// TIA Portal project "Vyrobne_kleman_Omdrejka_1.1" (V15.1)

(* hardware
DEVICE "S7-1200 station_1"  S7-1200 Station
   slot 0: "Rack_0"  S7-1200 Rack  Rack  V1.0
   slot 1: "PLC_1"  CPU 1215C DC/DC/DC  6ES7 215-1AG40-0XB0  V4.2
*)

// ===== PLC "PLC_1"  CPU 1215C DC/DC/DC =====

VAR_GLOBAL   // PLC tag table "dig_IN"
   "KS1_VZ" AT %I0.0 : Bool;   // posuvnik 1 zadne TL
   "KS1_VP" AT %I0.1 : Bool;
   "KS2_VP" AT %I0.2 : Bool;
   "KS2_VZ" AT %I0.3 : Bool;
   "OS1" AT %I0.4 : Bool;
   "OS2" AT %I0.5 : Bool;
   "T_LOAD" AT %I0.6 : Bool;
   "OS3" AT %I0.7 : Bool;
   "OS4" AT %I1.0 : Bool;
END_VAR

VAR_GLOBAL   // PLC tag table "dig_OUT"
   "P1_VZ" AT %Q0.0 : Bool;
   "P1_VP" AT %Q0.1 : Bool;
   "P2_VP" AT %Q0.2 : Bool;
   "P2_VZ" AT %Q0.3 : Bool;
   "D1" AT %Q0.4 : Bool;
   "D2" AT %Q0.5 : Bool;
   "S1" AT %Q0.6 : Bool;
   "D3" AT %Q0.7 : Bool;
   "S2" AT %Q1.0 : Bool;
   "D4" AT %Q1.1 : Bool;
END_VAR

VAR_GLOBAL   // PLC tag table "pomocne_premenne"
   "Pos_START" AT %M0.0 : Bool;
   "Pos1" AT %M0.1 : Bool;
   "Pos2" AT %M0.2 : Bool;
   "Pos3" AT %M0.3 : Bool;
   "Pos4" AT %M0.4 : Bool;
   "PosP" AT %M0.7 : Bool;
   "S1_pracuje" AT %M1.0 : Bool;
   "S1_dopracoval" AT %M1.1 : Bool;
   "S2_pracuje" AT %M1.3 : Bool;
   "S2_dopracoval" AT %M1.4 : Bool;
   "PosStart_id" AT %MW4 : Int;   // ID na zaciatku D1 po potvrdeni nalozenia
   "Pos1_id" AT %MW6 : Int;   // ID na linke 0 = prazdne
   "PosP_id" AT %MW8 : Int;   // ID na linke 0 = prazdne
   "Pos2_id" AT %MW10 : Int;   // ID na linke 0 = prazdne
   "Pos3_id" AT %MW12 : Int;   // ID na linke 0 = prazdne
   "Pos4_id" AT %MW14 : Int;   // ID na linke 0 = prazdne
   "Ptrig_1" AT %M20.0 : Bool;   // T_LOAD
   "Ptrig_2" AT %M20.1 : Bool;   // prerusenie OS1
   "Ptrig_3" AT %M20.2 : Bool;   // prerusenie OS2
   "Ptrig_4" AT %M20.3 : Bool;   // reset_CTU_1
   "ptrig_5" AT %M20.5 : Bool;   // OS3
   "ptrig_6" AT %M20.6 : Bool;   // Reset_CTU_S2
   "ptrig_7" AT %M20.7 : Bool;   // OS4
   "ptrig_8" AT %M21.0 : Bool;   // krok_1
   "ptrig_9" AT %M21.1 : Bool;   // pos_4==2
   "ptrig_10" AT %M21.2 : Bool;   // krok_4
   "ptrig_11" AT %M21.3 : Bool;   // posStart_r
   "ptrig_12" AT %M21.4 : Bool;   // pos1_r
   "ptrig_13" AT %M21.5 : Bool;   // posp_r
   "ptrig_14" AT %M21.6 : Bool;   // pos2_r
   "ptrig_15" AT %M21.7 : Bool;   // pos3_r
   "krok" AT %MW22 : Int;   // cislo kroku triedenia
END_VAR

DATA_BLOCK "DB_premenne"   // DB12
{ S7_Optimized_Access := 'TRUE' }
VERSION : 0.1
   VAR RETAIN
      ID_objekt : Int := 1;
      S1_cyklus : Int := 2;
      S2_cyklus : Int := 2;
   END_VAR
BEGIN
END_DATA_BLOCK

// folder: System blocks/Program resources

DATA_BLOCK "IEC_Timer_0_DB"   // DB1
{ S7_Optimized_Access := 'TRUE' }
AUTHOR : Simatic
FAMILY : IEC
NAME : IEC_TMR
VERSION : 1.0
// stored: InstanceOfName IEC_TIMER
"IEC_TIMER"
BEGIN
END_DATA_BLOCK

DATA_BLOCK "casovac_D1_na_PosP"   // DB2
{ S7_Optimized_Access := 'TRUE' }
AUTHOR : Simatic
FAMILY : IEC
NAME : IEC_TMR
VERSION : 1.0
// stored: InstanceOfName IEC_TIMER
"IEC_TIMER"
BEGIN
END_DATA_BLOCK

DATA_BLOCK "IEC_Timer_0_DB_1"   // DB3
{ S7_Optimized_Access := 'TRUE' }
AUTHOR : Simatic
FAMILY : IEC
NAME : IEC_TMR
VERSION : 1.0
// stored: InstanceOfName IEC_TIMER
"IEC_TIMER"
BEGIN
END_DATA_BLOCK

DATA_BLOCK "timer_S2_S"   // DB4
{ S7_Optimized_Access := 'TRUE' }
AUTHOR : Simatic
FAMILY : IEC
NAME : IEC_TMR
VERSION : 1.0
// stored: InstanceOfName IEC_TIMER
"IEC_TIMER"
BEGIN
END_DATA_BLOCK

DATA_BLOCK "timer_S2_R"   // DB5
{ S7_Optimized_Access := 'TRUE' }
AUTHOR : Simatic
FAMILY : IEC
NAME : IEC_TMR
VERSION : 1.0
// stored: InstanceOfName IEC_TIMER
"IEC_TIMER"
BEGIN
END_DATA_BLOCK

DATA_BLOCK "Rpocet_cyklov2"   // DB6
{ S7_Optimized_Access := 'TRUE' }
AUTHOR : Simatic
FAMILY : IEC
NAME : CNTR
VERSION : 1.0
// stored: InstanceOfName IEC_COUNTER
"IEC_COUNTER"
BEGIN
END_DATA_BLOCK

DATA_BLOCK "Rpocet_cyklov1"   // DB7
{ S7_Optimized_Access := 'TRUE' }
AUTHOR : Simatic
FAMILY : IEC
NAME : CNTR
VERSION : 1.0
// stored: InstanceOfName IEC_COUNTER
"IEC_COUNTER"
BEGIN
END_DATA_BLOCK

DATA_BLOCK "IEC_Timer_0_DB_2"   // DB8
{ S7_Optimized_Access := 'TRUE' }
AUTHOR : Simatic
FAMILY : IEC
NAME : IEC_TMR
VERSION : 1.0
// stored: InstanceOfName IEC_TIMER
"IEC_TIMER"
BEGIN
END_DATA_BLOCK

DATA_BLOCK "IEC_Timer_0_DB_3"   // DB9
{ S7_Optimized_Access := 'TRUE' }
AUTHOR : Simatic
FAMILY : IEC
NAME : IEC_TMR
VERSION : 1.0
// stored: InstanceOfName IEC_TIMER
"IEC_TIMER"
BEGIN
END_DATA_BLOCK

DATA_BLOCK "IEC_Timer_0_DB_4"   // DB10
{ S7_Optimized_Access := 'TRUE' }
AUTHOR : Simatic
FAMILY : IEC
NAME : IEC_TMR
VERSION : 1.0
// stored: InstanceOfName IEC_TIMER
"IEC_TIMER"
BEGIN
END_DATA_BLOCK

DATA_BLOCK "IEC_Timer_0_DB_5"   // DB11
{ S7_Optimized_Access := 'TRUE' }
AUTHOR : Simatic
FAMILY : IEC
NAME : IEC_TMR
VERSION : 1.0
// stored: InstanceOfName IEC_TIMER
"IEC_TIMER"
BEGIN
END_DATA_BLOCK

// folder: (top level)

ORGANIZATION_BLOCK "Main"   // OB1, LAD, ProgramCycle
TITLE = "Main Program Sweep (Cycle)"
{ S7_Optimized_Access := 'TRUE' }
VERSION : 0.1
   VAR_INPUT
      Initial_Call : Bool;   // Initial call of this OB
      Remanence : Bool;   // =True, if remanent data are available
   END_VAR
   VAR_TEMP   // added for the SCL form of the ladder/FBD networks
      _w1 : Bool;
      _w2 : Bool;
      _w3 : Bool;
      _w4 : Bool;
      _w5 : Bool;
      _w6 : Bool;
      _w7 : Bool;
      _w8 : Bool;
      _w9 : Bool;
   END_VAR
BEGIN

REGION Network 1: D1 nalozenie
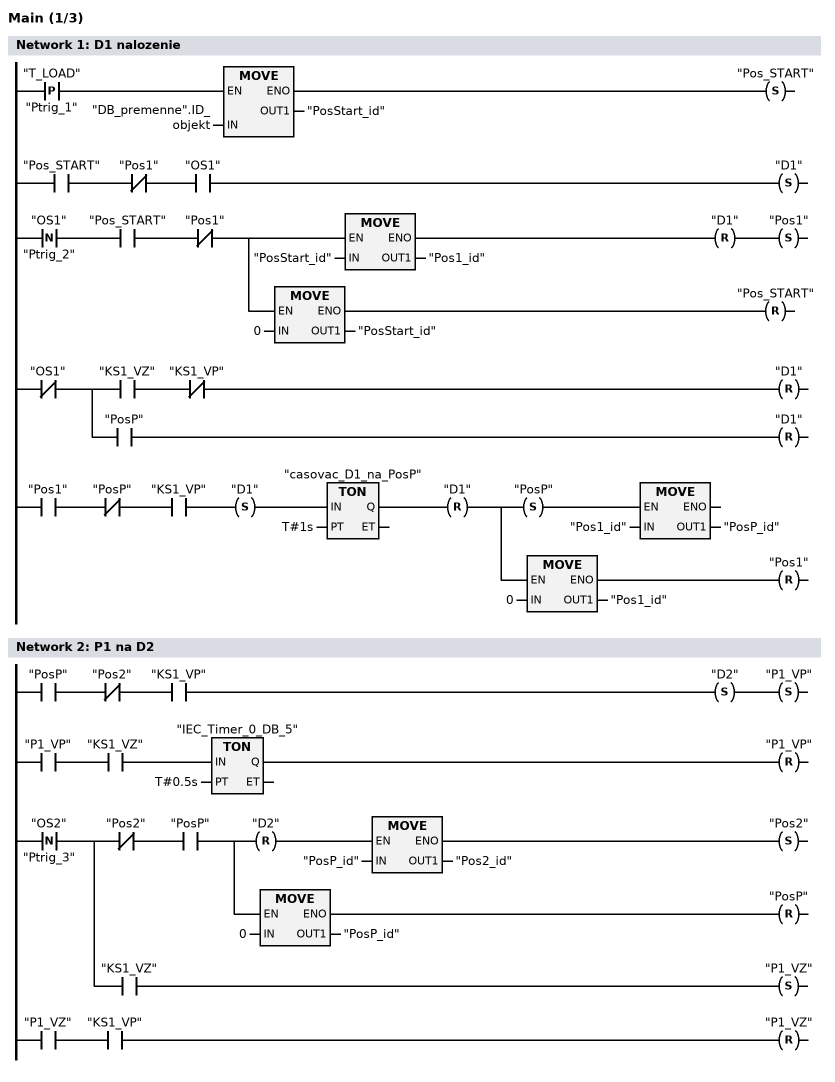
   #_w1 := "T_LOAD" AND NOT "Ptrig_1";   // rising edge of "T_LOAD"
   "Ptrig_1" := "T_LOAD";
   IF #_w1 THEN
       "PosStart_id" := "DB_premenne".ID_objekt;
       "Pos_START" := TRUE;
   END_IF;
   IF "Pos_START" AND NOT "Pos1" AND "OS1" THEN "D1" := TRUE; END_IF;
   #_w2 := NOT "OS1" AND "Ptrig_2";   // falling edge of "OS1"
   "Ptrig_2" := "OS1";
   IF #_w2 AND "Pos_START" AND NOT "Pos1" THEN
       "Pos1_id" := "PosStart_id";
       "D1" := FALSE;
   END_IF;
   #_w3 := #_w2 AND "Pos_START" AND NOT "Pos1";
   IF #_w3 THEN
       "Pos1" := TRUE;
       "PosStart_id" := 0;
       "Pos_START" := FALSE;
   END_IF;
   IF NOT "OS1" AND "KS1_VZ" AND NOT "KS1_VP" THEN "D1" := FALSE; END_IF;
   IF NOT "OS1" AND "PosP" THEN "D1" := FALSE; END_IF;
   #_w4 := "Pos1" AND NOT "PosP" AND "KS1_VP";
   IF #_w4 THEN "D1" := TRUE; END_IF;
   "casovac_D1_na_PosP".TON(IN := #_w4, PT := T#1s);
   IF "casovac_D1_na_PosP".Q THEN
       "D1" := FALSE;
       "PosP" := TRUE;
       "PosP_id" := "Pos1_id";
       "Pos1_id" := 0;
       "Pos1" := FALSE;
   END_IF;
END_REGION

REGION Network 2: P1 na D2
   IF "PosP" AND NOT "Pos2" AND "KS1_VP" THEN
       "D2" := TRUE;
       "P1_VP" := TRUE;
   END_IF;
   "IEC_Timer_0_DB_5".TON(IN := "P1_VP" AND "KS1_VZ", PT := T#0.5s);
   IF "IEC_Timer_0_DB_5".Q THEN "P1_VP" := FALSE; END_IF;
   #_w1 := NOT "OS2" AND "Ptrig_3";   // falling edge of "OS2"
   "Ptrig_3" := "OS2";
   IF #_w1 AND NOT "Pos2" AND "PosP" THEN
       "D2" := FALSE;
       "Pos2_id" := "PosP_id";
   END_IF;
   #_w2 := #_w1 AND NOT "Pos2" AND "PosP";
   IF #_w2 THEN
       "Pos2" := TRUE;
       "PosP_id" := 0;
       "PosP" := FALSE;
   END_IF;
   IF #_w1 AND "KS1_VZ" THEN "P1_VZ" := TRUE; END_IF;
   IF "P1_VZ" AND "KS1_VP" THEN "P1_VZ" := FALSE; END_IF;
END_REGION

REGION Network 3: S1
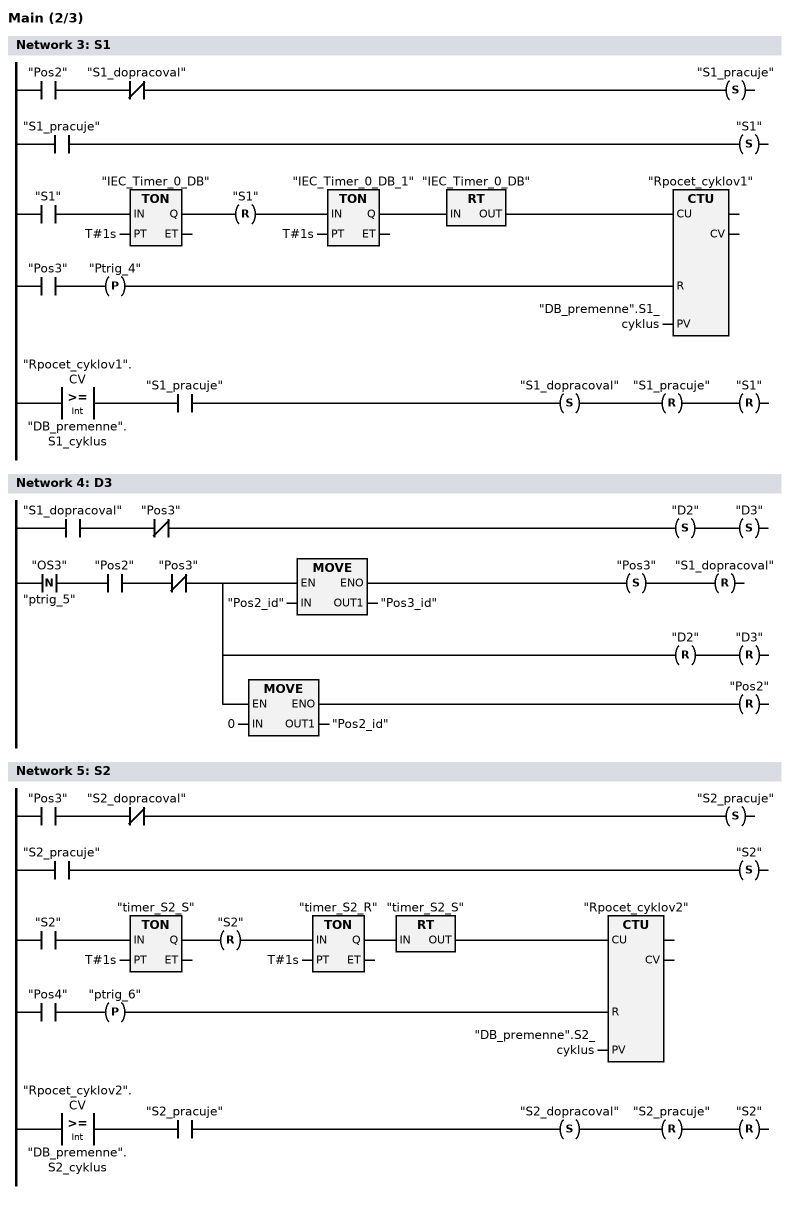
   IF "Pos2" AND NOT "S1_dopracoval" THEN "S1_pracuje" := TRUE; END_IF;
   IF "S1_pracuje" THEN "S1" := TRUE; END_IF;
   "IEC_Timer_0_DB".TON(IN := "S1", PT := T#1s);
   IF "IEC_Timer_0_DB".Q THEN "S1" := FALSE; END_IF;
   "IEC_Timer_0_DB_1".TON(IN := "IEC_Timer_0_DB".Q, PT := T#1s);
   IF "IEC_Timer_0_DB_1".Q THEN RESET_TIMER("IEC_Timer_0_DB"); END_IF;
   #_w1 := "Pos3" AND NOT "Ptrig_4";   // rising edge
   "Ptrig_4" := "Pos3";
   "Rpocet_cyklov1".CTU(CU := "IEC_Timer_0_DB_1".Q, R := #_w1, PV := "DB_premenne".S1_cyklus);
   IF ("Rpocet_cyklov1".CV >= "DB_premenne".S1_cyklus) AND "S1_pracuje" THEN "S1_dopracoval" := TRUE; END_IF;
   #_w2 := ("Rpocet_cyklov1".CV >= "DB_premenne".S1_cyklus) AND "S1_pracuje";
   IF #_w2 THEN
       "S1_pracuje" := FALSE;
       "S1" := FALSE;
   END_IF;
END_REGION

REGION Network 4: D3
   RUNG wire#powerrail
      Contact( "S1_dopracoval" )
      I_Contact( "Pos3" )
      S_Coil( "D2" )
      S_Coil( "D3" )
   END_RUNG
   RUNG wire#powerrail
      N_Contact(operand := "OS3", bit := "ptrig_5")
      Contact( "Pos2" )
      I_Contact( "Pos3" )
      wire#w1
      Move(in := "Pos2_id", out1 => "Pos3_id")
      S_Coil( "Pos3" )
      R_Coil( "S1_dopracoval" )
   END_RUNG
   RUNG wire#w1
      R_Coil( "D2" )
      R_Coil( "D3" )
   END_RUNG
   RUNG wire#w1
      Move(in := 0, out1 => "Pos2_id")
      R_Coil( "Pos2" )
   END_RUNG
   // the same network as SCL:
   IF "S1_dopracoval" AND NOT "Pos3" THEN
       "D2" := TRUE;
       "D3" := TRUE;
   END_IF;
   #_w1 := NOT "OS3" AND "ptrig_5";   // falling edge of "OS3"
   "ptrig_5" := "OS3";
   IF #_w1 AND "Pos2" AND NOT "Pos3" THEN "Pos3_id" := "Pos2_id"; END_IF;
   #_w2 := #_w1 AND "Pos2" AND NOT "Pos3";
   IF #_w2 THEN
       "Pos3" := TRUE;
       "S1_dopracoval" := FALSE;
       "D2" := FALSE;
       "D3" := FALSE;
       "Pos2_id" := 0;
       "Pos2" := FALSE;
   END_IF;
END_REGION

REGION Network 5: S2
   IF "Pos3" AND NOT "S2_dopracoval" THEN "S2_pracuje" := TRUE; END_IF;
   IF "S2_pracuje" THEN "S2" := TRUE; END_IF;
   "timer_S2_S".TON(IN := "S2", PT := T#1s);
   IF "timer_S2_S".Q THEN "S2" := FALSE; END_IF;
   "timer_S2_R".TON(IN := "timer_S2_S".Q, PT := T#1s);
   IF "timer_S2_R".Q THEN RESET_TIMER("timer_S2_S"); END_IF;
   #_w1 := "Pos4" AND NOT "ptrig_6";   // rising edge
   "ptrig_6" := "Pos4";
   "Rpocet_cyklov2".CTU(CU := "timer_S2_R".Q, R := #_w1, PV := "DB_premenne".S2_cyklus);
   IF ("Rpocet_cyklov2".CV >= "DB_premenne".S2_cyklus) AND "S2_pracuje" THEN "S2_dopracoval" := TRUE; END_IF;
   #_w2 := ("Rpocet_cyklov2".CV >= "DB_premenne".S2_cyklus) AND "S2_pracuje";
   IF #_w2 THEN
       "S2_pracuje" := FALSE;
       "S2" := FALSE;
   END_IF;
END_REGION

REGION Network 6: D4
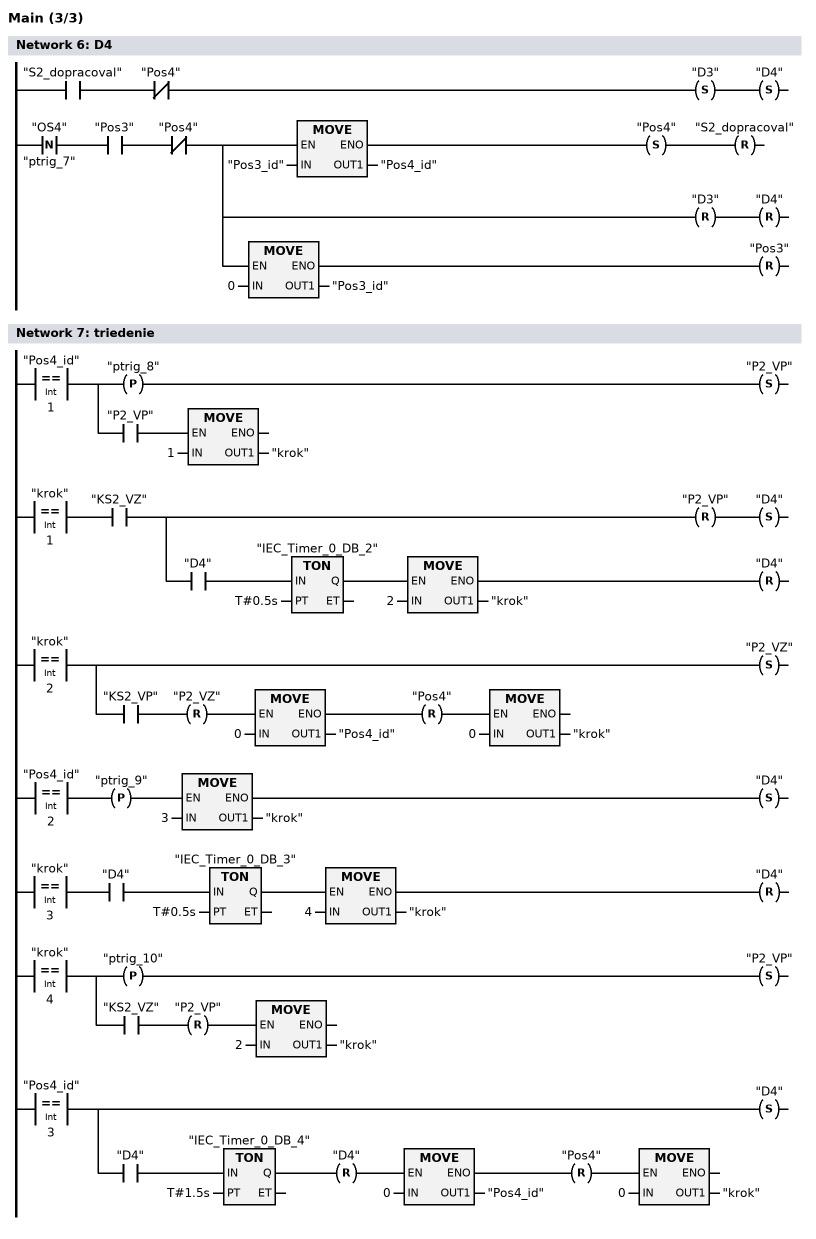
   RUNG wire#powerrail
      Contact( "S2_dopracoval" )
      I_Contact( "Pos4" )
      S_Coil( "D3" )
      S_Coil( "D4" )
   END_RUNG
   RUNG wire#powerrail
      N_Contact(operand := "OS4", bit := "ptrig_7")
      Contact( "Pos3" )
      I_Contact( "Pos4" )
      wire#w1
      Move(in := "Pos3_id", out1 => "Pos4_id")
      S_Coil( "Pos4" )
      R_Coil( "S2_dopracoval" )
   END_RUNG
   RUNG wire#w1
      R_Coil( "D3" )
      R_Coil( "D4" )
   END_RUNG
   RUNG wire#w1
      Move(in := 0, out1 => "Pos3_id")
      R_Coil( "Pos3" )
   END_RUNG
   // the same network as SCL:
   IF "S2_dopracoval" AND NOT "Pos4" THEN
       "D3" := TRUE;
       "D4" := TRUE;
   END_IF;
   #_w1 := NOT "OS4" AND "ptrig_7";   // falling edge of "OS4"
   "ptrig_7" := "OS4";
   IF #_w1 AND "Pos3" AND NOT "Pos4" THEN "Pos4_id" := "Pos3_id"; END_IF;
   #_w2 := #_w1 AND "Pos3" AND NOT "Pos4";
   IF #_w2 THEN
       "Pos4" := TRUE;
       "S2_dopracoval" := FALSE;
       "D3" := FALSE;
       "D4" := FALSE;
       "Pos3_id" := 0;
       "Pos3" := FALSE;
   END_IF;
END_REGION

REGION Network 7: triedenie
   #_w1 := "Pos4_id" = 1;
   #_w2 := #_w1 AND NOT "ptrig_8";   // rising edge
   "ptrig_8" := #_w1;
   IF #_w2 THEN "P2_VP" := TRUE; END_IF;
   IF #_w1 AND "P2_VP" THEN "krok" := 1; END_IF;
   #_w3 := ("krok" = 1) AND "KS2_VZ";
   IF #_w3 THEN
       "P2_VP" := FALSE;
       "D4" := TRUE;
   END_IF;
   "IEC_Timer_0_DB_2".TON(IN := #_w3 AND "D4", PT := T#0.5s);
   IF "IEC_Timer_0_DB_2".Q THEN
       "krok" := 2;
       "D4" := FALSE;
   END_IF;
   #_w4 := "krok" = 2;
   IF #_w4 THEN "P2_VZ" := TRUE; END_IF;
   IF #_w4 AND "KS2_VP" THEN
       "P2_VZ" := FALSE;
       "Pos4_id" := 0;
       "Pos4" := FALSE;
       "krok" := 0;
   END_IF;
   #_w5 := "Pos4_id" = 2;
   #_w6 := #_w5 AND NOT "ptrig_9";   // rising edge
   "ptrig_9" := #_w5;
   IF #_w6 THEN
       "krok" := 3;
       "D4" := TRUE;
   END_IF;
   "IEC_Timer_0_DB_3".TON(IN := ("krok" = 3) AND "D4", PT := T#0.5s);
   IF "IEC_Timer_0_DB_3".Q THEN
       "krok" := 4;
       "D4" := FALSE;
   END_IF;
   #_w7 := "krok" = 4;
   #_w8 := #_w7 AND NOT "ptrig_10";   // rising edge
   "ptrig_10" := #_w7;
   IF #_w8 THEN "P2_VP" := TRUE; END_IF;
   IF #_w7 AND "KS2_VZ" THEN
       "P2_VP" := FALSE;
       "krok" := 2;
   END_IF;
   #_w9 := "Pos4_id" = 3;
   IF #_w9 THEN "D4" := TRUE; END_IF;
   "IEC_Timer_0_DB_4".TON(IN := #_w9 AND "D4", PT := T#1.5s);
   IF "IEC_Timer_0_DB_4".Q THEN
       "D4" := FALSE;
       "Pos4_id" := 0;
       "Pos4" := FALSE;
       "krok" := 0;
   END_IF;
END_REGION
END_ORGANIZATION_BLOCK